Yaskawa INFORM job: TESTMIRROR.JBI

/JOB
//NAME TESTMIRROR
//POS
///NPOS 5,5,5,0,0,0
///TOOL 0
///POSTYPE PULSE
///PULSE
C00000=-146986,-745,-53104,-60690,90268,-28355
C00001=-152328,2483,-5521,-60971,72721,-18223
C00002=-154958,-7968,-4058,-61372,63554,-12173
C00003=-155055,-9564,-9245,-61661,69050,-17066
C00004=-146986,-745,-53104,-60690,90268,-28355
BC00000=64145,843878,573298
BC00001=54890,786548,810543
BC00002=54890,786548,810543
BC00003=66494,858426,513092
BC00004=64145,843878,573298
EC00000=266053,2
EC00001=266051,1
EC00002=354737,0
EC00003=266053,0
EC00004=266053,2
//INST
///DATE 2024/06/25 14:52
///ATTR SC,RW
///GROUP1 RB1,BS1
///GROUP2 ST1
NOP
MOVJ C00000 BC00000 VJ=25.00  +MOVJ EC00000 VJ=0.78
MOVJ C00001 BC00001 VJ=25.00  +MOVJ EC00001 VJ=0.78
SMOVL C00002 BC00002 V=100.0  +MOVJ EC00002
SMOVL C00003 BC00003 V=100.0  +MOVJ EC00003
MOVJ C00004 BC00004 VJ=25.00  +MOVJ EC00004 VJ=0.78
END
